Staubli VAL3: cmdDisableVolt.pgx

public program cmdDisableVolt(num x_nAxNum)
begin
  //"Disable voltage"字段无效
  doFaultReset[x_nAxNum]=false
  doEnableVoltage[x_nAxNum]=false
end
